(* PLC project  *)

PROGRAM BlocksXml
  VAR
    A : INT;
  END_VAR

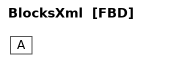
(* FBD diagram, written out as Structured Text *)
(* drawn but not wired to any output: A *)
END_PROGRAM
